{attribute 'qualified_only'}
VAR_GLOBAL CONSTANT
    {attribute 'analysis' := '-33'}      // Disable SA0033: Unused variable
    StringBuilder_MaxStringLength : UINT := 1024;
END_VAR

(* stored: Version 1.1.0.1
   GVL GVL_Param_AUT_Utilities: Id {a1668b94-fa3c-453e-a051-af918792153b}, ParameterList True *)
